VAR CONSTANT
	    CstClockReadTime 		: LTIME := LTIME#1S;	  				// (Time) Read Modbus Frequency .	
END_VAR

METHOD M_Execute
//////////////////
//  Method Calls 
/////////////////

VAR 
	// Method local variables (reinitialized at each cycle) 

END_VAR
SUPER^.M_Execute();
END_METHOD

END_FUNCTION_BLOCK

// ---- 01_Equipement_Library/ProtectRelay/FB_ProtectRelay_SepamS48.TcPOU
FUNCTION_BLOCK FB_ProtectRelay_SepamS48 EXTENDS FB_ProtectRelay_Base
//////////////////
// SEPAM system for High Voltage or Low Voltage Grid Protection. 
//////////////////

VAR_INPUT PERSISTENT
	// Parameters of the Object (instance/model specific) 
	   ParamTimeoutRTU						: TIME  := T#10S;					(* (s)	  Com RTU Timeout *)
	   ParamUnitID							: BYTE 	:= 1;						(* (NA)	  unit ID*)
	   ParamInInterfaceSub					: BOOL;								(* (NA)   Serial interface RS422/RS485 TYPE (0:EL6021, 1:SUB9)*)
END_VAR

VAR_OUTPUT
	//Child objects
	OUT_Protect_GTE_LONG_Running			: BOOL; 							// Long GTE fault, PP stop for 2m and lost of autorisation 

END_VAR

VAR_INPUT
	// I/O Inputs	
	IN_MesAlarmIMax_IO						: BOOL; 							// I max fault Fault, Losing autorisation and not possible to consumed
	IN_MesAlarmUmin_IO						: BOOL; 							// U min Fault, Keeping autorisation, If we have 3 gte in 30 min ==> Stop fedding and consumed during 2h
	IN_MesAlarmPWH_IO						: BOOL; 							// Defaut wattmétrique
	                                                								                                                	
	IN_CmdReset_3GTEFault					: BOOL; 							// 3GTE Fault Reset 
		
END_VAR

VAR
	//M_Read
	Trig_Read								: R_TRIG;
	ModbusRTU								: FB_ModbusRTU ;					// (NA) FB for Modbus Reading
	MbStruct								: ARRAY[1..2] OF Struct_InputRTU;

                                			
	ModbusAlarm								: ARRAY[1..2] OF BOOL;					// (NA) Read alarm
	AX_Quantity								: ARRAY[1..2] OF WORD;					// (NA) Quantity of blocks to read
	AX_Address								: ARRAY[1..2] OF WORD;					// (NA) Start address of the read
	OutErrorMbRead							: ARRAY[1..2] OF BOOL;
                                			
	Busy									: BOOL;
	MesBlock_Temp							: ARRAY [1..2] OF ARRAY [0..94] OF WORD;
	                            			
	RTrigI									: R_TRIG;
MesDataExd					AT %Q* 		: ProtectRelay_S48  ; 
	                            			
	//M_EVALUATE                			
	TON_GteIsLong							: TON;


		
END_VAR

METHOD M_Execute
//////////////////
//  Method Calls 
/////////////////

VAR 
	// Method local variables (reinitialized at each cycle) 
	MesStateCB	 : BOOL;

	KK 			 : INT;
	CalNbFeederClosed	: UINT ; 
END_VAR



CalNbFeederClosed := 0 ; 
FOR KK:= 1 TO CstNbFeederMVCB_G DO 
	CalNbFeederClosed :=  CalNbFeederClosed + SEL(A1_SUBMV.AX_FeederMVCB[KK].MesClosed , 0, 1 ) ; 

END_FOR




	
MesStateCB := A1_SUBMV.A1_MainMVCB.MesDataExd.MesData.MesClosed;
MesDataExd.MesData.MesI1 := 0;

IF MesStateCB THEN
	FOR KK:=1 TO CstNbPTR_G DO
	MesDataExd.MesData.MesI1 := MesDataExd.MesData.MesI1 + AX_PTR[KK].MesDataExd.MesData.MesI;
	END_FOR  
	

MesDataExd.MesData.MesI1 := MesDataExd.MesData.MesI1 *CalNbFeederClosed /CstNbFeederMVCB_G;
		

	
MesDataExd.MesData.MesI2 	:= MesDataExd.MesData.MesI1 ; 	
MesDataExd.MesData.MesI3 	:= MesDataExd.MesData.MesI1 ; 
MesDataExd.MesData.MesI0 	:= 0 ;
 
ELSE 
MesDataExd.MesData.MesI1 	:= 0 ;
MesDataExd.MesData.MesI2 	:= 0 ;
MesDataExd.MesData.MesI3 	:= 0 ;
MesDataExd.MesData.MesI0 	:= 0 ;
END_IF

MesDataExd.MesData.MesImax1	:= MAX(MesDataExd.MesData.MesImax1 , MesDataExd.MesData.MesI1  ) ; 
MesDataExd.MesData.MesImax2	:= MAX(MesDataExd.MesData.MesImax2 , MesDataExd.MesData.MesI2  ) ; 
MesDataExd.MesData.MesImax3	:= MAX(MesDataExd.MesData.MesImax3 , MesDataExd.MesData.MesI3  ) ; 
MesDataExd.MesData.MesImax0	:= MAX(MesDataExd.MesData.MesImax0 , MesDataExd.MesData.MesI0  ) ; 

MesDataExd.MesData.MesU12:= A1_SUBMV.MesDataExd.MesData.MesU;
MesDataExd.MesData.MesU31:= MesDataExd.MesData.MesU12;
MesDataExd.MesData.MesU23:= MesDataExd.MesData.MesU12;

MesDataExd.MesV1 := MesDataExd.MesData.MesU12/SQRT(3) ;
MesDataExd.MesV2 := MesDataExd.MesV1;	 
MesDataExd.MesV3 := MesDataExd.MesV1;

MesDataExd.MesData.MesFreq := A1_SUBMV.MesDataExd.MesData.MesFreq;
MesDataExd.MesP := A1_SUBMV.MesDataExd.MesData.MesPsol ; // Psol - Pload - Paux 
MesDataExd.MesQ := A1_SUBMV.MesDataExd.MesData.MesQsol; 
MesDataExd.MesS := SQRT(MesDataExd.MesP* MesDataExd.MesP + MesDataExd.MesQ*MesDataExd.MesQ);
MesDataExd.MesCosPhi := MesDataExd.MesP / MesDataExd.MesS;

IF MesDataExd.MesP > 0 THEN
	MesDataExd.EActProd := MesDataExd.EActProd + MesDataExd.MesP*ParamCycleTime_Emul/3600000	;
END_IF
IF MesDataExd.MesP < 0 THEN
	MesDataExd.EActCons := MesDataExd.EActCons - MesDataExd.MesP*ParamCycleTime_Emul/3600000	;
END_IF
IF MesDataExd.MesQ > 0 THEN
	MesDataExd.EReactProd := MesDataExd.EReactProd + MesDataExd.MesQ*ParamCycleTime_Emul/3600000	;
END_IF
IF MesDataExd.MesQ < 0 THEN
	MesDataExd.EReactCons := MesDataExd.EReactCons - MesDataExd.MesQ*ParamCycleTime_Emul/3600000	;
END_IF
END_METHOD

END_FUNCTION_BLOCK

// ---- 01_Equipement_Library/ProtectRelay/FB_ProtectRelay_SepamT20.TcPOU
FUNCTION_BLOCK FB_ProtectRelay_SepamT20 EXTENDS FB_ProtectRelay_Base
//////////////////
// SEPAM system for High Voltage or Low Voltage Grid Protection . 
//////////////////
VAR_INPUT PERSISTENT
	// Parameters of the Object (instance/model specific) 
	 
END_VAR

VAR_OUTPUT
	//Child objects
	OutFBCompleteted						: BOOL;
END_VAR

VAR_INPUT
	InUnitID            : DINT;			// (NA)   ID FOR SEPAM T20 Modbus Unit ID. 

	// I/O Inputs		
END_VAR

VAR
	//M_Read
	FB_ModbusRead_I1						: FB_ReadModbusRTU_V2; 				// (NA) FB for Modbus Reading
	FB_ModbusRead_I2						: FB_ReadModbusRTU_V2; 				// (NA) FB for Modbus Reading
	FB_ModbusRead_I3						: FB_ReadModbusRTU_V2; 				// (NA) FB for Modbus Reading
	ParamTimeoutRTU							: TIME:=T#10S;
	MesBlock1_Temp							: ARRAY [0..36] OF WORD;
	MesBlock2_Temp							: WORD;
	MesBlock3_Temp							: WORD;
	MesModbusAlarmCode						: UDINT;							// (NA) Modbus Read Alarm Code
	MesModbusAlarmCode2						: UDINT;							// (NA) Modbus Read Alarm Code
	MesModbusAlarmCode3						: UDINT;							// (NA) Modbus Read Alarm Code
	ModbusReadAlarm 						: BOOL;								// (NA) Modbus Read Alarm for communications
	ModbusReadAlarm2 						: BOOL;	
	ModbusReadAlarm3 						: BOOL;	
	AX_bRead 								: ARRAY [1..3] OF BOOL;
	CalAllCompleted							: BOOL;
	//M_ALARMMANAGEMENT VARIABLES//

	//M_Execute
	AllNotBusy								: BOOL;
	TP_Read									: TP;
	RTrig									: R_TRIG;
//	ClockRead								: BOOL;
	
	//EValuate//
MesDataExd					AT %Q* 		: ProtectRelay_T20;
	

		
END_VAR

METHOD M_Execute
//////////////////
//  Method Calls 
/////////////////

VAR 
	// Method local variables (reinitialized at each cycle) 

END_VAR
SUPER^.M_Execute();
END_METHOD

END_FUNCTION_BLOCK

// ---- 01_Equipement_Library/ProtectRelay/FB_ProtectRelay_VIP410.TcPOU
FUNCTION_BLOCK FB_ProtectRelay_VIP410 EXTENDS FB_ProtectRelay_Base
//////////////////
// SEPAM system for High Voltage or Low Voltage Grid Protection . 
//////////////////
VAR_INPUT PERSISTENT
	ParamTcpPort				: UINT:=502;    // (NA) TCP port
	ParamIPAddress				: STRING; 		// (NA) IP address
	ParamUnitID					: BYTE; 		// (NA) unit ID
END_VAR

VAR_OUTPUT
	
END_VAR

VAR_INPUT
		IN_MesTrip_IO			: BOOL ; 
END_VAR

VAR
	
	MesDataExd		AT %Q* 		: ProtectRelay_VIP410;
	FB_ModbusRead	          	: ARRAY[1..4] OF FB_ModbusRead; 
	ClockReadInput				: BOOL;

	MesBlock1_Temp 				: ARRAY [1..1] OF WORD ; 
	MesBlock2_Temp 				: ARRAY [1..20] OF WORD ; 
	MesBlock3_Temp 				: ARRAY [1..8] OF WORD ; 
	MesBlock4_Temp 				: ARRAY [1..2] OF WORD ; 
	AX_ModbusReadAlarm			: ARRAY[1..4] OF BOOL;
	AX_ModbusReadAlarmId		: ARRAY[1..4] OF UDINT;	
//	TP1							: TP ; 				// (NA) Tempo to define Modbus Reading Frequency 
	ParamClockInputTime 		: TIME 		:= TIME#5S;	  		// (Time) Read Modbus Frequency . 
END_VAR

METHOD M_Execute
//////////////////
//  Method Calls 
/////////////////

VAR 
	// Method local variables (reinitialized at each cycle) 

END_VAR
SUPER^.M_Execute();
END_METHOD

END_FUNCTION_BLOCK

// ---- 01_Equipement_Library/ProtectRelay/FB_ProtectRelay_WIP1.TcPOU
FUNCTION_BLOCK FB_ProtectRelay_WIP1 EXTENDS FB_ProtectRelay_Base
VAR_INPUT
						
	
	

END_VAR

VAR_INPUT
	// I/O Inputs 		                                     				
		IN_MesAlarmImax_IO		: BOOL ; // IO max I  fault
		IN_MesAlarmUmin_IO		: BOOL ;  // IO Min U  Fault 
		
END_VAR


VAR
// M_ALARMMNGMT VARIABLES //
                            		
	CmdResetHVCell				: BOOL ; 
	// M_READ VARIABLES//
	
MesDataExd 		    AT %Q*  	: ProtectRelay_WIP1; 	
		


END_VAR

METHOD M_Execute
SUPER^.M_Execute();
END_METHOD

END_FUNCTION_BLOCK

// ---- 01_Equipement_Library/Router/FB_Router.TcPOU
FUNCTION_BLOCK FB_Router

VAR_INPUT PERSISTENT 
	ParamTempoRestart	: TIME 		:= T#30S ;	//  (s)Tempo to wait before resupplying the ADSL routeur

	
END_VAR

        	
VAR_INPUT           	
	Heure_Local     	: TIMESTRUCT;
	IN_CmdRestart 			: BOOL;

	
	IN_CmdReset_L			: BOOL ;	// (NA) External Reset Command
	
END_VAR     


VAR_OUTPUT
	//Child objects
		OUT_CmdOpen_IO			: BOOL;	
END_VAR        	
      	
VAR                 	
	bInit				: BOOL;	// Booleen d'initialisation
		
	TP_Restart			: TP;
	// State Mananger //
	
	MesState			: BYTE; // Cal
MesDataExd			: Router_Standard;
	// M_Evaluate //
	
END_VAR

METHOD M_Execute : BOOL
VAR_INPUT
END_VAR
END_METHOD

END_FUNCTION_BLOCK

// ---- 01_Equipement_Library/Sensors/ANA/FB_ANA_Base.TcPOU
FUNCTION_BLOCK FB_ANA_Base 
//////////////////
// Analogic sensor . Base FB . 
//////////////////

VAR_INPUT PERSISTENT
	// Parameters of the Object (instance/mùodel specific) 
	ParamVarMaxAlarm		: REAL 		:=105		; // (%)  Config : Maximal allowed Site Hygrometry 
	ParamVarMaxWarning		: REAL 		:=90		; // (%)  Config : Maximal Site hygrometry warning
	ParamVarMinAlarm		: REAL 		:=-5		; // (%)  Config : Minimal allowed Site Hygrometry 
	ParamVarMinWarning		: REAL 		:=0			; // (%)  Config : Minimal Site hygrometry warning
	ParamDiffMax			: REAL 		:= 20 ; 	; // (NA) Config : Maximal Analogic difference acceptable between two sensors
	
	ParamNbSensors			: INT 		:=1			; // (NA) Config : Number of sensors
	
END_VAR

VAR_OUTPUT
	//Child objects
	
END_VAR

VAR_INPUT
	// I/O Inputs 
		IN_MesValue1_IO					: INT ; 	// 	IO Value
		IN_MesValue2_IO					: INT ; 	// 	IO Value

		IN_MesVar1Fault_IO		AT %I*		: BOOL ; 		 	//(NA)  sensor 1 has a 0 mA fault . 
		IN_MesVar2Fault_IO				: BOOL ; 		 	//(NA)  sensor 2 has a 0 mA fault . 		
END_VAR

VAR
	//M_ALARMMANAGEMENT VARIABLES//

		RS_MaxAlarm: RS;
		RS_MinAlarm: RS;
		RS_MinWarning: RS;
		RS_MaxWarning: RS;
	
		RSDiff: RS;
                                         	
	//M_READ VARIABLES//
		MesValue1						: REAL ;  	// temporary Value
		MesValue2						: REAL ; 
		
//	MesDataExd					: ANA ; 
	//EMULATOR //
		
		// M_INIT //
		bInit 						: BOOL;
		IN_CmdReset_L					: BOOL;
END_VAR

METHOD M_Execute
//////////////////
//  Method Calls 
/////////////////

VAR 
	// Method local variables (reinitialized at each cycle) 

END_VAR
END_METHOD

END_FUNCTION_BLOCK

// ---- 01_Equipement_Library/Sensors/ANA/FB_ANA_IO.TcPOU
FUNCTION_BLOCK FB_ANA_IO EXTENDS FB_ANA_Base
//////////////////
// Analogic sensor . Base FB . 
//////////////////

VAR_INPUT PERSISTENT
	// Parameters of the Object (instance/mùodel specific) 
		ParamName				: STRING:='TempPcs' ;			// (NA) Name of the pyranometer : to easily identify it
		ParamScaleMin			: REAL:=4 ; 		// (NA) minimal input value . 
		ParamScaleMax			: REAL:=20 ; 		// (NA) maximal input value .
		ParamRangeMin			: REAL:=0 ; 		// (NA) minimal output value . Unit depends on output 
		ParamRangeMax			: REAL:=100 ; 		// (NA) maximal output value . Unit depends on output 

		
		ParamForced_4_20		: BOOL:=FALSE;		// Is the input between 4-20mA ? 
		ParamPT100				: BOOL:=FALSE;	// IF PT 100
		ParamFix				: INT:=1 ; // Value to wich divide the initial value 
END_VAR

VAR_OUTPUT
	//Child objects
	
END_VAR

VAR_INPUT
	// I/O Inputs 
		//MesIO1							: INT ; 	// 	IO Value
		IN_MesIOReal1						: REAL;
		IN_MesIOReal2						: REAL;
		
END_VAR

VAR
	//M_ALARMMANAGEMENT VARIABLES//
              MesData			: ANA ;     	
	//M_READ VARIABLES//


		
END_VAR

END_FUNCTION_BLOCK

// ---- 01_Equipement_Library/Sensors/ANA/FB_ANA_Irra_Fx.TcPOU
FUNCTION_BLOCK FB_ANA_Irra_Fx EXTENDS FB_ANA_Base
//////////////////
// (4-20 mA) sensor . 
//////////////////

VAR_INPUT PERSISTENT
	// Parameters of the Object (instance/model specific) 
	ParamSensibility				: REAL ;			// Sensibility of the sensor ? 
END_VAR

VAR_OUTPUT
	//Child objects
	
END_VAR

VAR_INPUT
	// I/O Inputs 
	
END_VAR         			
                			
VAR             			
	A						: REAL;     // F(x) = Ax+B
	B						: REAL;     // F(x) = Ax+B

	 MesData			: ANA ;   
		
END_VAR

METHOD M_Execute
//////////////////
//  Method Calls 
/////////////////

VAR 
	// Method local variables (reinitialized at each cycle) 

END_VAR


SUPER^.M_Execute() ;
END_METHOD

END_FUNCTION_BLOCK

// ---- 01_Equipement_Library/Sensors/COM/FB_AllInOne.TcPOU
FUNCTION_BLOCK FB_AllInOne
VAR_INPUT
	ParamNameAllInOne		: STRING 	:= 'Wind spd + dir + hygro + temp';				// (NA) Name of the pyranometer : to easily identify it
	ParamTempoComAlarm		: TIME 		:= T#10S ; 										// (s) Config : Tempo to detect LOC Alarm
	ParamClockReadTime 		: TIME 		:= T#2S;	  									// (Time) Read Modbus Frequency . 
 	ParamTimeout			: TIME  	:= T#5S ;		  								// (Time) Timeout for modbus reading
	ParamUnitID				: BYTE		:= 1;											// (NA) Unit ID for modbus reading
	ParamTCPPort			: UINT		:= 502;											// (NA) TCP port for modbus
	ParamIpAddress			: STRING	:= '127.0.0.1';									// (NA) IP address for modbus
END_VAR

VAR
	//M_AlarmManagement
	TON_ComAlarm				: TON ; 						// Tempo before deteting loss of communication. 

	
	IN_CmdReset_L					: BOOL;                                                        	
		
	// M_READ VARIABLES//
MesData		AT %Q*  : AllInOne ; 							// (NA) [P,H,B] INV  Data Structure 
	FB_ModbusReadInputRegs		: ARRAY[1..2] OF FB_MBReadInputRegs;		// FB for Modbus Read
	MesBlock1_Temp 				: ARRAY[1..96]  OF WORD; 		// (NA) Temporary Block with multiple modbus reading (Caution : Double Word variables)
	MesBlock2_Temp 				: ARRAY[1..3]  OF WORD; 		// (NA) Temporary Block with multiple modbus reading (Caution : Double Word variables)
	MesModbusReadAlarm1 		: BOOL ; 						// (NA) Modbus Read Alarm for all modbus frames		
	MesModbusReadAlarm2 		: BOOL ; 						// (NA) Modbus Read Alarm for all modbus frames		
	MesAlarmCom					: BOOL;
	MesModbusAlarmCode			: UDINT;						// (NA) Modbus Read Alarm Code	
	
	// M_STATEMANAGER//
	FB_OperationIndex			: FB_OperationIndex ; 
	CalLastStart				: STRING ;			 			// Datetime of the last Start
	MesState					: BYTE ; 						// (NA) Cal                                                                                                            	
	CalRunningTime				: INT ; 						// Total Running Time
	                                                        	
	//M_EXECUTE VARIABLES //                                	
	TP1							: TP ; 							// (NA) Tempo to define Modbus Reading Frequency 
	                                                        	
	ClockRead					: BOOL;							// (NA) Modbus reading Clock
	
	
	//M_INIT //
	bInit 						: BOOL;							 
END_VAR

VAR_OUTPUT
END_VAR
VAR
END_VAR

METHOD M_Execute
//////////////////
//  Method Calls 
/////////////////

VAR 
	// Method local variables (reinitialized at each cycle) 

END_VAR
END_METHOD

END_FUNCTION_BLOCK

// ---- 01_Equipement_Library/Sensors/COM/FB_ANA_SMP1X.TcPOU
FUNCTION_BLOCK FB_ANA_SMP1X
VAR_INPUT PERSISTENT
	
	ParamNamePyranometer	: STRING 	:= 'Wind spd + dir + hygro + temp + pluvio';	// (NA) Name of the eqt : to easily identify it
	ParamTempoComAlarm		: TIME 		:= T#10S ; 										// (s) Config : Tempo to detect LOC Alarm
	ParamClockReadTime 		: TIME 		:= TIME#1S;	  									// (Time) Read Modbus Frequency . 
 	ParamTimeout			: TIME  	:= T#2S ;		  								// (Time) Timeout for modbus reading
	ParamUnitID				: BYTE		:= 1;											// (NA) Unit ID for modbus reading
	
END_VAR

VAR
	//M_AlarmManagement
	TON_ComAlarm				: TON ; 						// Tempo before deteting loss of communication. 

	MesAlarmCom					: BOOL;
	
	IN_CmdReset_L					: BOOL;                                                        	

	
	// M_READ VARIABLES//
		MesDataExd.MesData	AT %Q*	      	: SMP1X ; 					// (NA) [P,H,B] INV  Data Structure 
	//ModbusRead_RTU				: FB_ReadModbusRTU_V2;			// FB for Modbus Read
	bReadError					: BOOL;
	bReadCompleted 				: BOOL;
	bReadBusy					: BOOL;
	InputStructRead 			: Struct_InputRTU;
	
	MesBlock1_Temp 				: ARRAY[1..125]  OF WORD; 		// (NA) Temporary Block with multiple modbus reading (Caution : Double Word variables)
	MesModbusReadAlarm 		  	: BOOL ; 						// (NA) Modbus Read Alarm for all modbus frames		
	MesModbusAlarmCode			: UDINT;						// (NA) Modbus Read Alarm Code	
	
	ScaleFactor					: REAL;
	BodyTemp					: REAL;
	StatusFlag					: REAL;
	
	// M_STATEMANAGER//
	FB_OperationIndex			: FB_OperationIndex ; 
	CalLastStart				: STRING ;			 			// Datetime of the last Start
	MesState					: BYTE ; 						// (NA)                                                                                                            	
	CalRunningTime				: INT ; 						// Total Running Time
	                                                        	
	//M_EXECUTE VARIABLES //                                	
	TP1							: TP ; 							// (NA) Tempo to define Modbus Reading Frequency 
	                                                        	
	ClockRead					: BOOL;							// (NA) Modbus reading Clock
	
	
	//M_INIT //
	bInit 						: BOOL;							 
END_VAR

VAR_OUTPUT
END_VAR
VAR
END_VAR

METHOD M_Execute
//////////////////
//  Method Calls 
/////////////////

VAR 
	// Method local variables (reinitialized at each cycle) 

END_VAR
END_METHOD

END_FUNCTION_BLOCK

// ---- 01_Equipement_Library/Sensors/TOR/FB_TOR_Base.TcPOU
FUNCTION_BLOCK FB_TOR_Base
//////////////////
//  Digital SensOR  Base FB . 
//////////////////

VAR_INPUT PERSISTENT
	// Parameters of the Object (instance/model specific) 
	ParamNbSensors			: INT 		:=1			; // (NA) Config : Number of sensors, If =9 Then sensor is bi-stable contactOR 
	ParamAtleastOne			: BOOL 		:= TRUE ;  // If TRUE, the output is true if at leat one of the sensor is active. Otherwise , the output is true only if both are active
	ParamCableCutSecurity	: BOOL		:=FALSE;	// FALSE = ALARM ; 
	
	CalCountAlarm			: UDINT 	:=0 ; // Count number of times the alarm has been triggered.
	
END_VAR

VAR_OUTPUT
	//Child objects
	
END_VAR

VAR_INPUT
	// I/O Inputs 		                                     				
		IN_MesState1_IO 					: BOOL;	 				// (NA) First  Smoke detector IO, IF bi-stable NC
		IN_MesState2_IO					: BOOL ; 				// (NA) Second Smoke detector IO, IF Bi-stable NO
		IN_CmdReset_L					: BOOL;				// LOCAL Reset Value For Alarms
		IN_ResetCounter 				: BOOL ; 			// Reset counter . 
END_VAR

VAR
	//M_ALARMMANAGEMENT VARIABLES//

	//STATE MANAGEMENT //
//	MesDataExd				: TOR ; 	
		R_TRIGAlarm					: R_TRIG  ; 

	// EMULATOR 
	
END_VAR

METHOD M_Execute
//////////////////
//  Method Calls 
/////////////////

VAR 
	// Method local variables (reinitialized at each cycle) 
	
END_VAR
END_METHOD

END_FUNCTION_BLOCK

// ---- 01_Equipement_Library/Sensors/TOR/FB_TOR_CB.TcPOU
FUNCTION_BLOCK FB_TOR_CB EXTENDS FB_TOR_Base
//////////////////
//  Door sensor system . State = True >> Door Closed .
//////////////////

VAR_INPUT PERSISTENT
	// Parameters of the Object (instance/model specific) 
		
		
END_VAR

VAR_OUTPUT
	//Child objects
	
END_VAR

VAR_INPUT
	// I/O Inputs 		                                     				
		
END_VAR

VAR
	//M_ALARMMANAGEMENT VARIABLES//
		
MesDataExd			: TOR_Standard ;  

	
END_VAR

END_FUNCTION_BLOCK

// ---- 01_Equipement_Library/Sensors/TOR/FB_TOR_DS.TcPOU
FUNCTION_BLOCK FB_TOR_DS EXTENDS FB_TOR_Base
//////////////////
//  Door sensor system . State = True >> Door Closed .
//////////////////

VAR_INPUT PERSISTENT
	// Parameters of the Object (instance/model specific) 
		ParamTempoDoorAlarm			: TIME := T#10S ;	// (s) Tempo for Door sensor alarm 
		
END_VAR

VAR_OUTPUT
	//Child objects
	
END_VAR

VAR_INPUT
	// I/O Inputs 		                                     				
		
END_VAR

VAR
	//M_ALARMMANAGEMENT VARIABLES//
		TON_Ouverture				: TON;				//(NA) Tempo to detect door opened for too long time . 
	MesDataExd			: TOR_Standard ;  



END_VAR

METHOD M_Execute
//////////////////
//  Method Calls 
/////////////////

VAR 
	// Method local variables (reinitialized at each cycle) 
	
END_VAR


SUPER^.M_Execute() ;
END_METHOD

END_FUNCTION_BLOCK

// ---- 01_Equipement_Library/Sensors/TOR/FB_TOR_ES.TcPOU
FUNCTION_BLOCK FB_TOR_ES EXTENDS FB_TOR_Base
//////////////////
//  Emergency stop system
//////////////////
VAR_INPUT PERSISTENT
	// Parameters of the Object (instance/model specific) 
	ParamTempoEs :TIME:=T#2S;	// (s) Tempo before raising an alarm
END_VAR

VAR_OUTPUT
	//Child objects
	
END_VAR

VAR_INPUT
	// I/O Inputs 		                                     				
		
	
END_VAR

VAR
	//M_ALARMMANAGEMENT VARIABLES//
		FB_PermAlarm				: SR ;					// (NA) FB to maintain emergency stop Alarm 
		TON_ES						: TON ; 
 
	//M_STATEMANAGER VARIABLES//
		MesDataExd			: TOR_Standard ;  	
	// EMULATOR //
		Emul_MesState1				: BOOL;
		Emul_MesState2				: BOOL;
		
END_VAR

METHOD M_Execute
//////////////////
//  Method Calls 
/////////////////

VAR 
	// Method local variables (reinitialized at each cycle) 

END_VAR

	
	IF ParamNbSensors = 9 THEN // Use of contactor bi-stable No and NC
		IN_MesState2_IO := NOT IN_MesState2_IO;
	END_IF
SUPER^.M_Execute() ;
END_METHOD

END_FUNCTION_BLOCK

// ---- 01_Equipement_Library/Sensors/TOR/FB_TOR_Fuse.TcPOU
FUNCTION_BLOCK FB_TOR_Fuse EXTENDS FB_TOR_Base
//////////////////
//  Smoke and Fire detection system with Typhoon triggering system. 
//////////////////
VAR_INPUT PERSISTENT
	// Parameters of the Object (instance/model specific) 
	ParamTempoFuse :TIME:=T#5S;//  (s)Tempo before raising an alarm
END_VAR

VAR_OUTPUT
	//Child objects
	
END_VAR

VAR_INPUT
	// I/O Inputs 		                                     				
		
	
END_VAR

VAR
	//M_ALARMMANAGEMENT VARIABLES//
		FB_PermAlarm				: SR ;					// (NA) FB to maintain Fire Alarm even if sensor stop detection (burn) .
 		TON_Fuse					: TON; 	
	//M_STATEMANAGER VARIABLES//
	MesDataExd			: TOR_Standard ;  

		
END_VAR

METHOD M_Execute
//////////////////
//  Method Calls 
/////////////////

VAR 
	// Method local variables (reinitialized at each cycle) 

END_VAR
// EMULATOR I/O //

	
	IF ParamNbSensors = 9 THEN // Use of contactor bi-stable No and NC
		IN_MesState2_IO := NOT IN_MesState2_IO;
	END_IF
SUPER^.M_Execute() ;
END_METHOD

END_FUNCTION_BLOCK

// ---- 01_Equipement_Library/Sensors/TOR/FB_TOR_MS.TcPOU
FUNCTION_BLOCK FB_TOR_MS EXTENDS FB_TOR_Base
//////////////////
//  Door sensor system . State = True >> Door Closed .
//////////////////

VAR_INPUT PERSISTENT
	// Parameters of the Object (instance/model specific) 
		ParamTempoDoorAlarm			: TIME := T#10S ;	// (S) Tempo for Door sensor alarm 
		
END_VAR

VAR_OUTPUT
	//Child objects
	
END_VAR

VAR_INPUT
	// I/O Inputs 		                                     				
		
END_VAR

VAR
	//M_ALARMMANAGEMENT VARIABLES//
		TP_Fermeture			: TP;				//(NA) Tempo to detect door opened for too long time . 
		RS_fermeture			: RS;
		
		MesDataExd			: TOR_Standard ;  
		


END_VAR

METHOD M_Execute
//////////////////
//  Method Calls 
/////////////////

VAR 
	// Method local variables (reinitialized at each cycle) 
	
END_VAR

SUPER^.M_Execute() ;
END_METHOD

END_FUNCTION_BLOCK

// ---- 01_Equipement_Library/Sensors/TOR/FB_TOR_Rain.TcPOU
FUNCTION_BLOCK FB_TOR_Rain EXTENDS FB_TOR_Base
//////////////////
//  Door sensor system . State = True >> Door Closed .
//////////////////

VAR_INPUT PERSISTENT
	// Parameters of the Object (instance/model specific) 
	
		
END_VAR

VAR_OUTPUT
	//Child objects
	
END_VAR

VAR_INPUT
	// I/O Inputs 		                                     				
	
    ParamVarHrWarning   : REAL:=8;  // Max of raining before warning mm of rain for last hour --> Mean it is raining a lot  Defaut value 8       
    ParamVarDayWarning  : REAL:=48; // max of raining before warning mm of rain for last day  --> Mean it rained a lot during 1 day defaut value 48
	ParamVarMinAlarm	: REAL 	:=-5		; // (%)  Config : Minimal allowed Site Hygrometry 
	
END_VAR

VAR
	MesDataExd			: TOR_Rain;

	//M_ALARMMANAGEMENT VARIABLES//
		WarningDay					: BOOL;
		WarningHr					: BOOL;
		WarningValue				: BOOL;
	
	//GET/SET PROPERTY MANAGEMENT//
	//M_Execute
		FB_AverageHr				: FB_Average; 	
	    FB_AverageDay               : FB_Average;
	    FB_AverageMonth             : FB_Average;
		CTUHr						: CTU;
		CTUDay						: CTU;
		CTUMonth					: CTU;
		Hour 						: INT;
		PluvioHr_Avg		        : REAL ; 
		PluvioDay_Avg		        : REAL ; 
		PluvioMonth_Avg		        : REAL ;     
		PluvioHr_Max		        : REAL;
		PluvioDay_Max		        : REAL ; 
		PluvioMonth_Max		        : REAL ; 
        PluvioHr					: REAL ; 
		PluvioDay					: REAL ; 
		PluvioMonth					: REAL ; 

	
	
END_VAR

METHOD M_Execute
//////////////////
//  Method Calls 
/////////////////

VAR 
	// Method local variables (reinitialized at each cycle) 
	
END_VAR
// EMULATOR I/O //

//MAIN CODE HERE
Hour 							:=CstCycleTime_G/1000/3600  ;                        

CTUHr   (CU:= MesDataExd.MesData.MesAlarmState , RESET :=  Hour MOD 1 = 0) ; 
CTUDay  (CU:= MesDataExd.MesData.MesAlarmState , RESET := Hour MOD 24 = 0 ) ; 
CTUMonth(CU:= MesDataExd.MesData.MesAlarmState , RESET := Hour MOD 24*30 = 0 ) ; 

PluvioHr_Max := SEL( Hour MOD 1 = 0  ,   PluvioHr_Max , PluvioHr_Max:= PluvioHr)  ; 
PluvioHr := CTUHr.CV  ; 

PluvioDay_Max := SEL( Hour MOD 24 = 0  ,   PluvioDay_Max , PluvioDay_Max:= PluvioDay)  ; 
PluvioDay := CTUDay.CV  ; 

PluvioMonth_Max := SEL( Hour MOD 24*30 = 0  ,   PluvioMonth_Max , PluvioMonth_Max:= PluvioMonth)  ; 
PluvioMonth := CTUMonth.CV  ; 


FB_AverageHr(ValueIn:=PluvioHr_Max  , WindowDuration := 24*3600*1000 , ValueOut => PluvioHr_Avg) ; 
FB_AverageDay(ValueIn:=PluvioDay_Max  , WindowDuration := 24*30*3600*1000 , ValueOut => PluvioDay_Avg) ; 
FB_AverageMonth(ValueIn:=PluvioMonth_Max  , WindowDuration := 24*365*3600*1000 , ValueOut => PluvioMonth_Avg) ;
//EVALUATE

MesDataExd.MesRainFall_LastHour 	:= PluvioHr;
MesDataExd.MesRainFall_LastDay		:= PluvioDay;
MesDataExd.MesRainFall_LastMonth	:= PluvioMonth;
MesDataExd.AvgmmHour		:= PluvioHr_Avg;
MesDataExd.AvgmmDay		:= PluvioDay_Avg;
MesDataExd.AvgmmMonth		:= PluvioMonth_Avg;


SUPER^.M_Execute();
END_METHOD

END_FUNCTION_BLOCK

// ---- 01_Equipement_Library/Sensors/TOR/FB_TOR_SD.TcPOU
FUNCTION_BLOCK FB_TOR_SD EXTENDS FB_TOR_Base
//////////////////
//  Smoke and Fire detection system with Typhoon triggering system. 
//////////////////
VAR_INPUT PERSISTENT
	// Parameters of the Object (instance/model specific) 
	ParamTempoFire :TIME:=T#2S;//  (s)Tempo before raising an alarm
END_VAR

VAR_OUTPUT
	//Child objects
	
END_VAR

VAR_INPUT
	// I/O Inputs 		                                     				
		
	
END_VAR

VAR
	//M_ALARMMANAGEMENT VARIABLES//
		FB_PermAlarm				: SR ;					// (NA) FB to maintain Fire Alarm even if sensor stop detection (burn) .
		TON_Fire					: TON ; 
 
	//M_STATEMANAGER VARIABLES//
		MesDataExd			: TOR_Standard ;  
		
		
END_VAR

METHOD M_Execute
//////////////////
//  Method Calls 
/////////////////

VAR 
	// Method local variables (reinitialized at each cycle) 

END_VAR

	IF ParamNbSensors = 9 THEN // Use of contactor bi-stable No and NC
		IN_MesState2_IO := NOT IN_MesState2_IO;
	END_IF
SUPER^.M_Execute() ;
END_METHOD

END_FUNCTION_BLOCK

// ---- 01_Equipement_Library/Sensors/TOR/FB_TOR_Spd.TcPOU
FUNCTION_BLOCK FB_TOR_Spd EXTENDS FB_TOR_Base
//////////////////
//  Smoke and Fire detection system with Typhoon triggering system. 
//////////////////
VAR_INPUT PERSISTENT
	// Parameters of the Object (instance/model specific) 
	ParamTempoEs :TIME:=T#5S;//  (s)Tempo before raising an alarm
END_VAR

VAR_OUTPUT
	//Child objects
	
END_VAR

VAR_INPUT
	// I/O Inputs 		                                     				
		
	
END_VAR

VAR
	//M_ALARMMANAGEMENT VARIABLES//
		FB_PermAlarm				: SR ;					// (NA) FB to maintain Fire Alarm even if sensor stop detection (burn) .
		TON_ES						: TON ; 
 
	//M_STATEMANAGER VARIABLES//
		MesDataExd			: TOR_Standard ;  

		
END_VAR

METHOD M_Execute
//////////////////
//  Method Calls 
/////////////////

VAR 
	// Method local variables (reinitialized at each cycle) 

END_VAR

	
	IF ParamNbSensors = 9 THEN // Use of contactor bi-stable No and NC
		IN_MesState2_IO := NOT IN_MesState2_IO;
	END_IF
SUPER^.M_Execute() ;
END_METHOD

END_FUNCTION_BLOCK

// ---- 01_Equipement_Library/Sensors/TOR/FB_TOR_Standard.TcPOU
FUNCTION_BLOCK FB_TOR_Standard EXTENDS FB_TOR_Base
//////////////////
//  Circuit Breaker
//////////////////

VAR_INPUT PERSISTENT
	// Parameters of the Object (instance/model specific) 
		
		
END_VAR

VAR_OUTPUT
	//Child objects
	
END_VAR

VAR_INPUT
	// I/O Inputs 		                                     				
		
END_VAR

VAR
	//M_ALARMMANAGEMENT VARIABLES//
		
MesDataExd			: TOR_Standard ;  

	
END_VAR

END_FUNCTION_BLOCK

// ---- 01_Equipement_Library/Sensors/TOR/FB_TOR_ToS.TcPOU
FUNCTION_BLOCK FB_TOR_ToS EXTENDS FB_TOR_Base
//////////////////
//  Technician on site selectOR   
//////////////////

VAR_INPUT PERSISTENT
	// Parameters of the Object (instance/model specific) 
	ParamTempoToSAlarm				: TIME := T#180M ; 	//(min) Tempo (2h30) after ToS without clear fault >> alarm 
	ParamTempoToSWarning			: TIME := T#120M ;  // (min) Tempo (2h) after ToS without clear fault  >> warning
END_VAR

VAR_OUTPUT
	//Child objects
	
END_VAR

VAR_INPUT
	// I/O Inputs 		                                     				
	
END_VAR

VAR
	//M_ALARMMANAGEMENT VARIABLES//
		TON 						: TON ;  			 // (NA) Calculate time since technician presence activation. 
		        
MesDataExd			: TOR_Standard ;                              			
	          	
	//GET/SET PROPERTY MANAGEMENT//
	
	//EMULATOR //
		Emul_MesState				: BOOL;
		
END_VAR

METHOD M_Execute
//////////////////
//  Method Calls 
/////////////////

VAR 
	// Method local variables (reinitialized at each cycle) 

END_VAR
// EMULATOR I/O //

SUPER^.M_Execute() ;
END_METHOD

END_FUNCTION_BLOCK

// ---- 01_Equipement_Library/Tariff Meter/FB_EM.TcPOU
FUNCTION_BLOCK FB_EM EXTENDS FB_EM_Base
//////////////////
// Measurement Solution. Base FB
//////////////////
VAR_INPUT PERSISTENT
	// Parameters of the Object (instance specific) 
		
	
END_VAR

VAR_OUTPUT
	//Child objects
	
END_VAR
VAR
	//M_ALARMMANAGEMENT VARIABLES//
		Eess: REAL;
	Eessinit	: REAL ; 
                             

	//M_INIT VARIABLES //
	
		
	// M_EXECUTE VARIABLES //
 		
	// M_Reset_L
		
                      
END_VAR

VAR_INPUT
		
END_VAR

METHOD M_Execute
//////////////////
//  Method Calls 
/////////////////
VAR 
	// Method local variables (reinitialized at each cycle) 
	// EMULATOR

	
END_VAR
Eess :=  Eess + ((A1_PP.MesDataExd.MesData.MesPbat + A1_SUBMV.MesDataExd.MesData.MesPaux)/6)*ParamCycleTime_Emul/3600000  ; 

MesPulseEactCons := FALSE ; 
IF Eess > Eessinit + ParamStepEactCons THEN	// every 10 kWh 
	MesPulseEactCons := TRUE ; 
	Eessinit := Eess ; 
END_IF
END_METHOD

END_FUNCTION_BLOCK

// ---- 01_Equipement_Library/Tariff Meter/FB_EM_Base.TcPOU
FUNCTION_BLOCK FB_EM_Base
//////////////////
// Measurement Solution. Base FB
//////////////////
VAR_INPUT PERSISTENT
	// Parameters of the Object (instance specific) 
		CmdInitialValues			: EM;
		ParamStepEactCons			: REAL := 10;					// kWh step for tariff meter
		ParamStepEactProd			: REAL := 10;                 // kWh step for tariff meter
		ParamStepEreactCons			: REAL := 10;                 // kVArh step for tariff meter
		ParamStepEreactProd			: REAL := 10;                 // kVArh step for tariff meter
		ParamEssNum					: UINT :=1 ; 					// ESS Num
END_VAR

VAR_INPUT
	//Child objects
		IN_CmdReset_L					: BOOL;													// (NA) Local reset of the alarms	
END_VAR
VAR
	//M_ALARMMANAGEMENT VARIABLES//
		TON_ComAlarm				: TON ; 												// Tempo before deteting loss of communication. 

	//M_INIT VARIABLES //
		bInit						: BOOL 				:= TRUE ; 							// (NA) Initialize object parameters at first cycle 
		
	// M_EXECUTE VARIABLES //
 //	MesDataExd			: EM;					// (NA) Structure of the Tariff Meter
		
	// M_EVALUATE VARIABLES //
		trig1 						: R_TRIG;												// (NA) Trigger for the pulses
		trig2 						: R_TRIG;												// (NA) Trigger for the pulses
		trig3 						: R_TRIG;												// (NA) Trigger for the pulses
		trig4 						: R_TRIG;												// (NA) Trigger for the pulses

                      
END_VAR

VAR_INPUT
		MesPulseEactCons			: BOOL;													// Pulse Input signal for the Active energy consumed measurement
		MesPulseEactProd			: BOOL;													// Pulse Input signal for the Active energy produced measurement
		MesPulseEreactCons			: BOOL;													// Pulse Input signal for the Reactive energy consumed measurement
		MesPulseEreactProd			: BOOL;													// Pulse Input signal for the Reactive energy produced measurement
END_VAR

METHOD M_Execute
//////////////////
//  Method Calls 
/////////////////
VAR 
	// Method local variables (reinitialized at each cycle) 
	// EMULATOR

	
END_VAR
END_METHOD

END_FUNCTION_BLOCK

// ---- 01_Equipement_Library/Tariff Meter/FB_EM_Pulse.TcPOU
FUNCTION_BLOCK FB_EM_Pulse EXTENDS FB_EM_Base
//////////////////
// Measurement Solution. Base FB
//////////////////
VAR_INPUT PERSISTENT
	// Parameters of the Object (instance specific) 
		
	
END_VAR

VAR_OUTPUT
	//Child objects
	
END_VAR
VAR
	//M_ALARMMANAGEMENT VARIABLES//
		FB_DetectFixedValue   : FB_DetectFixedValue ; 
        Eact_null    		  : REAL ;                                   								
		

	//M_INIT VARIABLES //
		MesDataExd			: EM_Standard ; 
		
	// M_EXECUTE VARIABLES //
 		
	// M_Reset_L
		
                      
END_VAR

VAR_INPUT
		
END_VAR

METHOD M_AlarmManagement
//////////////////
// Digiware measurement tool alarm and warning management
/////////////////

VAR 
	FB_AlarmCodeManager : FB_AlarmCodeManager ; 
END_VAR

FB_DetectFixedValue(IN_Addr := ADR(MesDataExd.MesData.MesEactCons) , IN_Size := SIZEOF(MesDataExd.MesData.MesEactCons) , IN_Duration :=T#3H , IN_EmptyStruct := ADR(Eact_null ) ); 

// ALARM CODE //
	FB_AlarmCodeManager(
		bAlarm1			:= MesDataExd.MesData.MesEActProd > 10 ,																			// Production measured			
		bAlarm2			:=FB_DetectFixedValue.OUT_bStatic 	,																	// Loss of communication with meter 
		bAlarm3			:=FALSE, 																								// 
		bAlarm4			:=FALSE, 																								// 
		bAlarm5			:=FALSE, 																								//
		bAlarm6			:=FALSE,        																						//
		bAlarm7			:=FALSE,        																						//
		bAlarm8			:=FALSE,        																						//
		bAlarm9			:=FALSE,        																						//
		bAlarm10		:=FALSE,        																						//
		bAlarm11		:=FALSE,        																						//
		bAlarm12		:=FALSE,        																						//
		bAlarm13		:=FALSE,        																						//
		bAlarm14		:=FALSE,        																						//
		bAlarm15		:=FALSE,        																						//
		wAlarmCode		=>MesDataExd.MesData.MesAlarmCode);

// WARNING CODE //

	FB_AlarmCodeManager(
		bAlarm1			:= FALSE ,										//  
		bAlarm2			:=FALSE, 										// 
		bAlarm3			:=FALSE, 										// 
		bAlarm4			:=FALSE, 										// 
		bAlarm5			:=FALSE, 										//
		bAlarm6			:=FALSE,        								//
		bAlarm7			:=FALSE,        								//
		bAlarm8			:=FALSE,        								//
		bAlarm9			:=FALSE,        								//
		bAlarm10		:=FALSE,        								//
		bAlarm11		:=FALSE,        								//
		bAlarm12		:=FALSE,        								//
		bAlarm13		:=FALSE,        								//
		bAlarm14		:=FALSE,        								//
		bAlarm15		:=FALSE,        								//
		wAlarmCode		=>MesDataExd.MesData.MesWarningCode);
			
// EVENT CODE //
	FB_AlarmCodeManager(
		bAlarm1			:= IN_CmdReset_L, 				// Reset command
		bAlarm2			:= FALSE, 						// 
		bAlarm3			:= FALSE, 						// 
		bAlarm4			:= FALSE, 						// 
		bAlarm5			:= FALSE, 						//
		bAlarm6			:= FALSE, 						//
		bAlarm7			:= FALSE,                       //
		bAlarm8			:= FALSE,                       //
		bAlarm9			:= FALSE,                       //
		bAlarm10		:= FALSE,                       //
		bAlarm11		:= FALSE,                       //
		bAlarm12		:= FALSE,                       //
		bAlarm13		:= FALSE,                       //
		bAlarm14		:= FALSE,                       //
		bAlarm15		:= FALSE,                       //
		wAlarmCode		=>MesDataExd.MesData.MesEventCode);
END_METHOD

METHOD M_Evaluate
VAR_INPUT
END_VAR

VAR
	TM_0 : EM_Standard;	// Empty structure
	OutTrig_Eac : BOOL;
	OutTrig_Eap : BOOL;
	OutTrig_Erc : BOOL;
	OutTrig_Erp : BOOL;
	bTest : BOOL;
END_VAR
IF CmdInitialValues.MesData.MesEactCons <> TM_0.MesData.MesEactCons OR CmdInitialValues.MesData.MesEActProd <> TM_0.MesData.MesEActProd OR CmdInitialValues.MesData.MesEReactCons <> TM_0.MesData.MesEReactCons OR CmdInitialValues.MesData.MesEReactProd <> TM_0.MesData.MesEReactProd THEN
MesDataExd:= CmdInitialValues;
	CmdInitialValues := TM_0 ;
END_IF

trig1(CLK := IN_MesPulseEactCons_IO, Q => OutTrig_Eac);
trig2(CLK := IN_MesPulseEactProd_IO, Q => OutTrig_Eap);
trig3(CLK:= IN_MesPulseEreactCons_IO, Q => OutTrig_Erc);
trig4(CLK:= IN_MesPulseEreactProd_IO, Q => OutTrig_Erp);

IF OutTrig_Eac THEN
MesDataExd.MesData.MesEactCons := MesDataExd.MesData.MesEactCons + ParamStepEactCons;
END_IF 

IF OutTrig_Eap THEN
MesDataExd.MesData.MesEActProd := MesDataExd.MesData.MesEActProd + ParamStepEactProd;
END_IF 

IF OutTrig_Erc THEN
MesDataExd.MesData.MesEReactCons := MesDataExd.MesData.MesEReactCons + ParamStepEreactCons;
END_IF 

IF OutTrig_Erp THEN
MesDataExd.MesData.MesEReactProd := MesDataExd.MesData.MesEReactProd + ParamStepEreactProd;
END_IF 

SUPER^.M_Evaluate();
END_METHOD

METHOD M_Init
VAR 
	InitialValues : EM_Standard ; 
END_VAR
MesDataExd := InitialValues ; 
bInit := FALSE ;
END_METHOD

END_FUNCTION_BLOCK

// ---- 01_Equipement_Library/Transfo/FB_Transfo_Base.TcPOU
FUNCTION_BLOCK FB_Transfo_Base
//////////////////
// High Voltage transformer with Transfo or DMCR detection . 
//////////////////

VAR_INPUT PERSISTENT
	// Parameters of the Object (instance/model specific) 

END_VAR

VAR_OUTPUT
	//Child objects
	
END_VAR

VAR_INPUT
		// Transfo

END_VAR

VAR
	//MesDataExd					: Transfo ; 
		
END_VAR

METHOD M_Execute
//////////////////
//  Method Calls 
/////////////////

VAR 
	// Method local variables (reinitialized at each cycle) 

END_VAR
END_METHOD

END_FUNCTION_BLOCK

// ---- 01_Equipement_Library/Transfo/FB_Transfo_HVCom.TcPOU
FUNCTION_BLOCK FB_Transfo_HVCom EXTENDS FB_Transfo_Base
//////////////////
// High Voltage transformer with Transfo or DMCR detection . 
//////////////////

VAR_INPUT PERSISTENT
	// Parameters of the Object (instance/model specific) 
	
END_VAR

VAR_OUTPUT
	//Child objects
	
END_VAR

VAR_INPUT

END_VAR

VAR
MesDataExd					: Transfo_HV ; 
		
END_VAR

END_FUNCTION_BLOCK

// ---- 01_Equipement_Library/Transfo/FB_Transfo_MV.TcPOU
FUNCTION_BLOCK FB_Transfo_MV EXTENDS FB_Transfo_Base
//////////////////
// High Voltage transformer with Transfo or DMCR detection . 
//////////////////

VAR_INPUT PERSISTENT
	// Parameters of the Object (instance/model specific) 

END_VAR

VAR_OUTPUT
	//Child objects
	
END_VAR

VAR_INPUT
		// Transfo
	IN_MesWarningTemp_IO				: BOOL ; 		// (NA) Warning Oil Temperature IO
	IN_MesAlarmTemp_IO					: BOOL ; 		// (NA) Alarm Oil Temperature   IO
	IN_MesAlarmGas_IO					: BOOL ; 		// (NA) Gas Alarm               IO
	IN_MesAlarmPressure_IO				: BOOL ; 		// (NA) Oil Pressure Alarm		IO
	IN_MesAlarmsSynthesis_IO			: BOOL ;        // (NA) Alarms synthesis        IO 
	
END_VAR

VAR
MesDataExd					: Transfo_MV ; 
	Emul_Alarm_Temp						: BOOL := FALSE;			
	Emul_Alarm_Synthesis				: BOOL := FALSE;
	
END_VAR

METHOD M_Execute
//////////////////
//  Method Calls 
/////////////////

VAR 
	// Method local variables (reinitialized at each cycle) 
	
END_VAR
 MesDataExd.MesData.MesAlarmTemp 			:= Emul_Alarm_Temp;			
MesDataExd.MesData.MesAlarmsSynthesis 		:= Emul_Alarm_Synthesis;
END_METHOD

END_FUNCTION_BLOCK

// ---- 01_Equipement_Library/Transfo/FB_Transfo_MVCom.TcPOU
FUNCTION_BLOCK FB_Transfo_MVCom EXTENDS FB_Transfo_Base

//////////////////
// High Voltage transformer with Transfo or DMCR detection . 
//////////////////

VAR_INPUT PERSISTENT
	// Parameters of the Object (instance/model specific) 
	
END_VAR

VAR_OUTPUT
	//Child objects
	
END_VAR

VAR_INPUT

	
END_VAR

VAR
MesDataExd					: Transfo_MV ; 
		
END_VAR

END_FUNCTION_BLOCK

// ---- 01_Equipement_Library/UPS/FB_UPS_Base.TcPOU
FUNCTION_BLOCK FB_UPS_Base
//////////////////
// UPS 
//////////////////
VAR_INPUT PERSISTENT
	// Parameters of the Object (instance/model specific) 
		ParamTimeOut				: TIME := T#2S;		//  (s)Modbus Timeout
		ParamClockReadTime			: TIME := T#1S;		// (s) Modbus Reading Frequency 
		ParamNC						: BOOL :=FALSE ; 	// False: TRUE = Closed , True : TRUE = opened

		
		ParamTempoComAlarm			: TIME := T#2S;		// (s)Tempo before raising a communication alarm
		ParamTempoComWarning		: TIME := T#1S;		// (s)Tempo before raising a communication warning
		ParamEBatt  				: REAL := 225; 		// (Wh) Emulateur : Ebat for 48V
END_VAR

VAR_OUTPUT
	//Child objects
		OUT_CmdRelance_IO			: BOOL;
END_VAR

VAR_INPUT
	// I/O Inputs
		IN_MesDischarging_IO		: BOOL;
		IN_MesBatLow_IO		   		: BOOL;
		IN_MesFault_IO				: BOOL;

		IN_CmdRelanceChargeur_IO	: BOOL;
		
		IN_CmdToggleRead			: BOOL;
		IN_CmdReset_L				: BOOL ; 
END_VAR

VAR
	//M_ALARMMANAGEMENT VARIABLES//
		TON_ComAlarm				: TON;
		TON_ComWarning				: TON;	

		MesWarningCom				: BOOL ; 			// (NA) [P,H] True if bad modbus communication 
			
	//M_READ//
//	MesDataExd					: UPS ; 

	//M_EXECUTE //
		TP1							: TP;

		ClockRead		AT %Q*		: BOOL;

		   		
    //M_CP VARIABLES//
		Trig_Cmd_Read				: R_TRIG;                                                                                        
                                                                                       
		CmdRelanceChargeur			: BOOL;
		CP_Relance					: BOOL;
		TP_Relance					: TP;
		ParamTP_Impulsion			: TIME:=T#5S;

	// EMULATOR //
	
		
END_VAR

METHOD M_Execute
//////////////////
//  Method Calls 
/////////////////

VAR 
	// Method local variables (reinitialized at each cycle) 

END_VAR
END_METHOD

END_FUNCTION_BLOCK

// ---- 01_Equipement_Library/UPS/FB_UPS_CXC.TcPOU
FUNCTION_BLOCK FB_UPS_CXC EXTENDS FB_UPS_Base
//////////////////
// UPS 
//////////////////
VAR_INPUT PERSISTENT
	// Parameters of the Object (instance/model specific) 

		ParamIPAddress				: STRING 	:= '192.168.20.66'; 	// (NA)Config: IP Adress of PV INverter
		ParamUnitID 				: BYTE  	:= 1; 			  		// (NA)   Modbus Unit ID. 
		ParamTCPPort				: UINT		:= 502;					// (NA) TCP port for modbus
		
END_VAR

VAR_OUTPUT
	//Child objects
	
END_VAR

VAR_INPUT
	// I/O Inputs
		IN_MesCbUPS_IO				: BOOL ; // 1 = opened. 
END_VAR

VAR
	//M_ALARMMANAGEMENT VARIABLES//

	//M_READ//
		MesDataExd						AT %Q*	: UPS_CXC ; 
		AX_ModbusRead		   		: ARRAY [1..2] OF FB_ModbusRead ; 					// (NA) FB for Modbus Reading
		ModbusReadInput				: FB_ModbusReadInput ; 		       
                                 
		MesBlock_Temp 				: ARRAY [1..2] OF ARRAY[1..120]  OF WORD; 			// (NA) Temporary Block with multiple modbus reading (Caution : Double Word variables)
		MesBlockInput				: ARRAY[1..1] OF BYTE ; 
		
	
	//M_EXECUTE //
		bInit: BOOL;
		
END_VAR

METHOD M_Execute
//////////////////
//  Method Calls 
/////////////////

VAR 
	// Method local variables (reinitialized at each cycle) 

END_VAR

IF bInit THEN
	bInit := FALSE ; 
MesDataExd.MesData.MesSoC := 50 ; 
END_IF

MesDataExd.MesIdc := 3 ; 

MesDataExd.MesUBatt := 47.5 ; 
IF MesDataExd.MesData.MesSoC >=100 THEN 
MesDataExd.MesData.MesIBatt := SEL(A1_SUBMV.A1_MainMVCB.MesDataExd.MesData.MesClosed , MesDataExd.MesData.MesIdc ,0   ) ; // can only be negative discharging 
ELSE
MesDataExd.MesData.MesIBatt :=  SEL(A1_SUBMV.A1_MainMVCB.MesDataExd.MesData.MesClosed , MesDataExd.MesData.MesIdc , 4   ) ;
END_IF
MesDataExd.MesSoC :=  MAX( 0 , MesDataExd.MesData.MesSoC  + 100.MesDataExd.MesData.MesIBatt*.MesDataExd.MesData.MesUBatt * 1/3600000 * ParamCycleTime_Emul / ParamEBatt ) ; 


MesDataExd.MesIload  := MesDataExd.MesData.MesIdc + MesDataExd.MesData.MesIBatt ; 

MesDataExd.MesUdc :=  SEL(A1_SUBMV.MesDataExd.MesData.A1_MainMVCB.MesDataExd.MesData.MesClosed  MesDataExd.MesData.MesUBatt , 48 ) ;; 
MesDataExd.MesUac	:= SEL(A1_SUBMV.MesDataExd.MesData.A1_MainMVCB.MesDataExd.MesData.MesClosed  ,0 , 230 ) ;

MesDataExd.MesData.MesBatteryLow := MesDataExd.MesData.MesSoC < 20 ; // Low battery capacity 
MesDataExd.MesData.MesDischarging := MesDataExd.MesData.MesIBatt < 0; 
MesDataExd.MesData.MesFaultSynthesis := MesDataExd.MesData.MesBatteryLow OR MesDataExd.MesData.MesDischarging ;
END_METHOD

END_FUNCTION_BLOCK

// ---- 01_Equipement_Library/UPS/FB_UPS_Eneris.TcPOU
FUNCTION_BLOCK FB_UPS_ENERIS EXTENDS FB_UPS_Base
//////////////////
// UPS 
//////////////////
VAR_INPUT PERSISTENT
	// Parameters of the Object (instance/model specific) 
	
END_VAR

VAR_OUTPUT
	//Child objects
	
END_VAR

VAR_INPUT
	// I/O Inputs
		IN_MesCbUPS_IO					: BOOL ; // 1 = opened. 
END_VAR

VAR
	//M_ALARMMANAGEMENT VARIABLES//
		
	//M_READ//

	MesDataExd				: UPS_ENERIS ; 
	
		
	//M_EXECUTE //
		
	
END_VAR

METHOD M_Execute
//////////////////
//  Method Calls 
/////////////////

VAR 
	// Method local variables (reinitialized at each cycle) 

END_VAR
END_METHOD

END_FUNCTION_BLOCK

// ---- 01_Equipement_Library/UPS/FB_UPS_PS10048.TcPOU
FUNCTION_BLOCK FB_UPS_PS10048 EXTENDS FB_UPS_Base
//////////////////
// SEPAM system for High Voltage or Low Voltage Grid Protection. 
//////////////////

VAR_INPUT 
	ParamTcpPort				: UINT:=502;
	ParamIPAddress				: STRING; 
	ParamUnitID					: BYTE; 
END_VAR

VAR_OUTPUT
	
END_VAR

VAR_INPUT

END_VAR

VAR
MesDataExd    	AT %Q*	: UPS_PS10048;
	FB_ModbusRead	          	: ARRAY[1..4] OF FB_ModbusRead; 
			
	MesBlock1_Temp 				: ARRAY [1..1] OF WORD; 
	MesBlock2_Temp 				: ARRAY [1..11] OF WORD; 
	MesBlock3_Temp 				: ARRAY [1..8] OF WORD; 
	MesBlock4_Temp 				: ARRAY [1..2] OF WORD; 
	
	AX_ModbusReadAlarm			: ARRAY[1..4] OF BOOL;
	AX_ModbusReadAlarmId		: ARRAY[1..4] OF UDINT;	
	
	//M_EXECUTE //
	bInit: BOOL;
	
	
	// Emulator 
	Emul_MesAlamCom 			: BOOL := FALSE;
	Emul_MesAlarm_AcLow			: BOOL := FALSE;
	Emul_MesAlarm_AcOff			: BOOL := FALSE;
	Emul_MesAlarm_Charger		: BOOL := FALSE;
	
END_VAR

METHOD M_Execute
//////////////////
//  Method Calls 
/////////////////

VAR_INPUT
	
END_VAR
VAR 
	MW					: FB_MergeWordsToFloat;
	MW_1				: FB_MergeWordsToDint;
END_VAR
	//COM
MesDataExd.MesData.MesAlarmCom 	:= Emul_MesAlamCom;
MesDataExd.MesData.MesCapacity_Nom 		:= ParamEBatt.MesDataExd.MesData.MesUdc_48V; 	
	
MesDataExd.MesData.MesUdc_12V 			:= 12;		 

MesDataExd.MesData.MesCapacity_Nom 		:= 37000;
	                                
    MesDataExd.MesData.MesAlarm_AcLow		:= Emul_MesAlarm_AcLow;
	 
IF bInit THEN
	bInit 				:= FALSE; 
MesDataExd.MesData.MesSoC 	:= 50; 
END_IF

MesDataExd.MesUBatt 	:= 47.5 ; 
IF MesDataExd.MesData.MesSoC 	>=100 THEN 
MesDataExd.MesData.MesIdc_Bat  := SEL(A1_SUBMV.A1_MainMVCB.MesDataExd.MesData.MesClosed , -.MesDataExd.MesData.MesIdc_12V , 0) ; 			// can only be negative discharging 
ELSE
MesDataExd.MesData.MesIdc_Bat :=  SEL(A1_SUBMV.A1_MainMVCB.MesDataExd.MesData.MesClosed , MesDataExd.MesData.MesIdc_12V , 4) ;
END_IF

MesDataExd.MesSoC	  				:=  MAX( 0, MesDataExd.MesData.MesSoC  + 100.MesDataExd.MesData.MesIdc_Bat*.MesDataExd.MesData.MesUBatt * 1/3600000 * ParamCycleTime_Emul / ParamEBatt); 
MesDataExd.MesUdc_48V 				:=  SEL(A1_SUBMV.A1_MainMVCB.MesDataExd.MesData.MesClosed, MesDataExd.MesData.MesUBatt, 48) ; 

MesDataExd.MesData.MesAlarm_Ulow  	:= MesDataExd.MesData.MesSoC < 20 ; // Low battery capacity 
MesDataExd.MesData.MesDischarging 	:= MesDataExd.MesData.MesIdc_Bat < 0; 
	
MesDataExd.MesAlarm_AcOff 			:= Emul_MesAlarm_AcOff;
MesDataExd.MesAlarm_AcLow 			:= Emul_MesAlarm_AcLow;
MesDataExd.MesFault_Charger			:= Emul_MesAlarm_Charger;

MesdataExd.MesFault_Minor   		:= MesDataExd.MesData.MesAlarm_AcLow OR MesDataExd.MesData.MesAlarm_Ulow ;
MesdataExd.MesFault_Major   		:= MesDataExd.MesData.MesSoC < 10 OR MesDataExd.MesData.MesAlarm_AcOff OR MesDataExd.MesData.MesFault_Charger;
mesdataexd.MesAlarm_GeneralOff		:= MesDataExd.MesData.MesAlarm_AcOff OR MesDataExd.MesData.MesSoC < 5;
END_METHOD

END_FUNCTION_BLOCK

// ---- 04_Application/ADS/ADS_Param.TcPOU
PROGRAM ADS_Param
VAR
END_VAR

SignalName[1]:='GVL_CFG.AX_PTR[1].A1_INV_Smartlogger.MesDataExd.MesData.;	bClockIO[1]:=FALSE;	Taille[1]:=SIZEOF(GVL_CFG.AX_PTR[1].A1_INV_Smartlogger.MesDataExd.MesData.;	Address[1]:=ADR(GVL_CFG.AX_PTR[1].A1_INV_Smartlogger.MesDataExd.MesData.;	ReadAdsType[1]:=FALSE;	WriteAdsType[1]:=TRUE;
SignalName[2]:='GVL_CFG.AX_PTR[2].A1_INV_Smartlogger.MesDataExd.MesData.;	bClockIO[2]:=FALSE;	Taille[2]:=SIZEOF(GVL_CFG.AX_PTR[2].A1_INV_Smartlogger.MesDataExd.MesData.;	Address[2]:=ADR(GVL_CFG.AX_PTR[2].A1_INV_Smartlogger.MesDataExd.MesData.;	ReadAdsType[2]:=FALSE;	WriteAdsType[2]:=TRUE;
SignalName[3]:='GVL_CFG.AX_PTR[3].A1_INV_Smartlogger.MesDataExd.MesData.;	bClockIO[3]:=FALSE;	Taille[3]:=SIZEOF(GVL_CFG.AX_PTR[3].A1_INV_Smartlogger.MesDataExd.MesData.;	Address[3]:=ADR(GVL_CFG.AX_PTR[3].A1_INV_Smartlogger.MesDataExd.MesData.;	ReadAdsType[3]:=FALSE;	WriteAdsType[3]:=TRUE;
SignalName[4]:='GVL_CFG.AX_PTR[4].A1_INV_Smartlogger.MesDataExd.MesData.;	bClockIO[4]:=FALSE;	Taille[4]:=SIZEOF(GVL_CFG.AX_PTR[4].A1_INV_Smartlogger.MesDataExd.MesData.;	Address[4]:=ADR(GVL_CFG.AX_PTR[4].A1_INV_Smartlogger.MesDataExd.MesData.;	ReadAdsType[4]:=FALSE;	WriteAdsType[4]:=TRUE;
SignalName[5]:='GVL_CFG.AX_PTR[1].A1_INV_Smartlogger.WriteBlock_Temp';	bClockIO[5]:=TRUE;	Taille[5]:=SIZEOF(GVL_CFG.AX_PTR[1].A1_INV_Smartlogger.WriteBlock_Temp);	Address[5]:=ADR(GVL_CFG.AX_PTR[1].A1_INV_Smartlogger.WriteBlock_Temp);	ReadAdsType[5]:=TRUE;	WriteAdsType[5]:=FALSE;
SignalName[6]:='GVL_CFG.AX_PTR[2].A1_INV_Smartlogger.WriteBlock_Temp';	bClockIO[6]:=TRUE;	Taille[6]:=SIZEOF(GVL_CFG.AX_PTR[2].A1_INV_Smartlogger.WriteBlock_Temp);	Address[6]:=ADR(GVL_CFG.AX_PTR[2].A1_INV_Smartlogger.WriteBlock_Temp);	ReadAdsType[6]:=TRUE;	WriteAdsType[6]:=FALSE;
SignalName[7]:='GVL_CFG.AX_PTR[3].A1_INV_Smartlogger.WriteBlock_Temp';	bClockIO[7]:=TRUE;	Taille[7]:=SIZEOF(GVL_CFG.AX_PTR[3].A1_INV_Smartlogger.WriteBlock_Temp);	Address[7]:=ADR(GVL_CFG.AX_PTR[3].A1_INV_Smartlogger.WriteBlock_Temp);	ReadAdsType[7]:=TRUE;	WriteAdsType[7]:=FALSE;
SignalName[8]:='GVL_CFG.AX_PTR[4].A1_INV_Smartlogger.WriteBlock_Temp';	bClockIO[8]:=TRUE;	Taille[8]:=SIZEOF(GVL_CFG.AX_PTR[4].A1_INV_Smartlogger.WriteBlock_Temp);	Address[8]:=ADR(GVL_CFG.AX_PTR[4].A1_INV_Smartlogger.WriteBlock_Temp);	ReadAdsType[8]:=TRUE;	WriteAdsType[8]:=FALSE;
SignalName[9]:='GVL_CFG.AX_PTR[1].A1_INV_Smartlogger.ClockRead';	bClockIO[9]:=TRUE;	Taille[9]:=SIZEOF(GVL_CFG.AX_PTR[1].A1_INV_Smartlogger.ClockRead);	Address[9]:=ADR(GVL_CFG.AX_PTR[1].A1_INV_Smartlogger.ClockRead);	ReadAdsType[9]:=TRUE;	WriteAdsType[9]:=FALSE;
SignalName[10]:='GVL_CFG.AX_PTR[2].A1_INV_Smartlogger.ClockRead';	bClockIO[10]:=TRUE;	Taille[10]:=SIZEOF(GVL_CFG.AX_PTR[2].A1_INV_Smartlogger.ClockRead);	Address[10]:=ADR(GVL_CFG.AX_PTR[2].A1_INV_Smartlogger.ClockRead);	ReadAdsType[10]:=TRUE;	WriteAdsType[10]:=FALSE;
SignalName[11]:='GVL_CFG.AX_PTR[3].A1_INV_Smartlogger.ClockRead';	bClockIO[11]:=TRUE;	Taille[11]:=SIZEOF(GVL_CFG.AX_PTR[3].A1_INV_Smartlogger.ClockRead);	Address[11]:=ADR(GVL_CFG.AX_PTR[3].A1_INV_Smartlogger.ClockRead);	ReadAdsType[11]:=TRUE;	WriteAdsType[11]:=FALSE;
SignalName[12]:='GVL_CFG.AX_PTR[4].A1_INV_Smartlogger.ClockRead';	bClockIO[12]:=TRUE;	Taille[12]:=SIZEOF(GVL_CFG.AX_PTR[4].A1_INV_Smartlogger.ClockRead);	Address[12]:=ADR(GVL_CFG.AX_PTR[4].A1_INV_Smartlogger.ClockRead);	ReadAdsType[12]:=TRUE;	WriteAdsType[12]:=FALSE;
SignalName[13]:='GVL_CFG.AX_PTR[1].A1_INV_Smartlogger.ClockWrite';	bClockIO[13]:=TRUE;	Taille[13]:=SIZEOF(GVL_CFG.AX_PTR[1].A1_INV_Smartlogger.ClockWrite);	Address[13]:=ADR(GVL_CFG.AX_PTR[1].A1_INV_Smartlogger.ClockWrite);	ReadAdsType[13]:=TRUE;	WriteAdsType[13]:=FALSE;
SignalName[14]:='GVL_CFG.AX_PTR[2].A1_INV_Smartlogger.ClockWrite';	bClockIO[14]:=TRUE;	Taille[14]:=SIZEOF(GVL_CFG.AX_PTR[2].A1_INV_Smartlogger.ClockWrite);	Address[14]:=ADR(GVL_CFG.AX_PTR[2].A1_INV_Smartlogger.ClockWrite);	ReadAdsType[14]:=TRUE;	WriteAdsType[14]:=FALSE;
SignalName[15]:='GVL_CFG.AX_PTR[3].A1_INV_Smartlogger.ClockWrite';	bClockIO[15]:=TRUE;	Taille[15]:=SIZEOF(GVL_CFG.AX_PTR[3].A1_INV_Smartlogger.ClockWrite);	Address[15]:=ADR(GVL_CFG.AX_PTR[3].A1_INV_Smartlogger.ClockWrite);	ReadAdsType[15]:=TRUE;	WriteAdsType[15]:=FALSE;
SignalName[16]:='GVL_CFG.AX_PTR[4].A1_INV_Smartlogger.ClockWrite';	bClockIO[16]:=TRUE;	Taille[16]:=SIZEOF(GVL_CFG.AX_PTR[4].A1_INV_Smartlogger.ClockWrite);	Address[16]:=ADR(GVL_CFG.AX_PTR[4].A1_INV_Smartlogger.ClockWrite);	ReadAdsType[16]:=TRUE;	WriteAdsType[16]:=FALSE;
SignalName[17]:='GVL_CFG.AX_PTR[1].AX_INV[1].MesDataExd.MesData.;	bClockIO[17]:=FALSE;	Taille[17]:=SIZEOF(GVL_CFG.AX_PTR[1].AX_INV[1].MesDataExd.MesData.;	Address[17]:=ADR(GVL_CFG.AX_PTR[1].AX_INV[1].MesDataExd.MesData.;	ReadAdsType[17]:=FALSE;	WriteAdsType[17]:=TRUE;
SignalName[18]:='GVL_CFG.AX_PTR[1].AX_INV[2].MesDataExd.MesData.;	bClockIO[18]:=FALSE;	Taille[18]:=SIZEOF(GVL_CFG.AX_PTR[1].AX_INV[2].MesDataExd.MesData.;	Address[18]:=ADR(GVL_CFG.AX_PTR[1].AX_INV[2].MesDataExd.MesData.;	ReadAdsType[18]:=FALSE;	WriteAdsType[18]:=TRUE;
SignalName[19]:='GVL_CFG.AX_PTR[2].AX_INV[1].MesDataExd.MesData.;	bClockIO[19]:=FALSE;	Taille[19]:=SIZEOF(GVL_CFG.AX_PTR[2].AX_INV[1].MesDataExd.MesData.;	Address[19]:=ADR(GVL_CFG.AX_PTR[2].AX_INV[1].MesDataExd.MesData.;	ReadAdsType[19]:=FALSE;	WriteAdsType[19]:=TRUE;
SignalName[20]:='GVL_CFG.AX_PTR[2].AX_INV[2].MesDataExd.MesData.;	bClockIO[20]:=FALSE;	Taille[20]:=SIZEOF(GVL_CFG.AX_PTR[2].AX_INV[2].MesDataExd.MesData.;	Address[20]:=ADR(GVL_CFG.AX_PTR[2].AX_INV[2].MesDataExd.MesData.;	ReadAdsType[20]:=FALSE;	WriteAdsType[20]:=TRUE;
SignalName[21]:='GVL_CFG.AX_PTR[3].AX_INV[1].MesDataExd.MesData.;	bClockIO[21]:=FALSE;	Taille[21]:=SIZEOF(GVL_CFG.AX_PTR[3].AX_INV[1].MesDataExd.MesData.;	Address[21]:=ADR(GVL_CFG.AX_PTR[3].AX_INV[1].MesDataExd.MesData.;	ReadAdsType[21]:=FALSE;	WriteAdsType[21]:=TRUE;
SignalName[22]:='GVL_CFG.AX_PTR[3].AX_INV[2].MesDataExd.MesData.;	bClockIO[22]:=FALSE;	Taille[22]:=SIZEOF(GVL_CFG.AX_PTR[3].AX_INV[2].MesDataExd.MesData.;	Address[22]:=ADR(GVL_CFG.AX_PTR[3].AX_INV[2].MesDataExd.MesData.;	ReadAdsType[22]:=FALSE;	WriteAdsType[22]:=TRUE;
SignalName[23]:='GVL_CFG.AX_PTR[4].AX_INV[1].MesDataExd.MesData.;	bClockIO[23]:=FALSE;	Taille[23]:=SIZEOF(GVL_CFG.AX_PTR[4].AX_INV[1].MesDataExd.MesData.;	Address[23]:=ADR(GVL_CFG.AX_PTR[4].AX_INV[1].MesDataExd.MesData.;	ReadAdsType[23]:=FALSE;	WriteAdsType[23]:=TRUE;
SignalName[24]:='GVL_CFG.AX_PTR[4].AX_INV[2].MesDataExd.MesData.;	bClockIO[24]:=FALSE;	Taille[24]:=SIZEOF(GVL_CFG.AX_PTR[4].AX_INV[2].MesDataExd.MesData.;	Address[24]:=ADR(GVL_CFG.AX_PTR[4].AX_INV[2].MesDataExd.MesData.;	ReadAdsType[24]:=FALSE;	WriteAdsType[24]:=TRUE;
SignalName[25]:='GVL_CFG.AX_PTR[1].AX_INV[1].ClockRead';	bClockIO[25]:=TRUE;	Taille[25]:=SIZEOF(GVL_CFG.AX_PTR[1].AX_INV[1].ClockRead);	Address[25]:=ADR(GVL_CFG.AX_PTR[1].AX_INV[1].ClockRead);	ReadAdsType[25]:=TRUE;	WriteAdsType[25]:=FALSE;
SignalName[26]:='GVL_CFG.AX_PTR[1].AX_INV[2].ClockRead';	bClockIO[26]:=TRUE;	Taille[26]:=SIZEOF(GVL_CFG.AX_PTR[1].AX_INV[2].ClockRead);	Address[26]:=ADR(GVL_CFG.AX_PTR[1].AX_INV[2].ClockRead);	ReadAdsType[26]:=TRUE;	WriteAdsType[26]:=FALSE;
SignalName[27]:='GVL_CFG.AX_PTR[2].AX_INV[1].ClockRead';	bClockIO[27]:=TRUE;	Taille[27]:=SIZEOF(GVL_CFG.AX_PTR[2].AX_INV[1].ClockRead);	Address[27]:=ADR(GVL_CFG.AX_PTR[2].AX_INV[1].ClockRead);	ReadAdsType[27]:=TRUE;	WriteAdsType[27]:=FALSE;
SignalName[28]:='GVL_CFG.AX_PTR[2].AX_INV[2].ClockRead';	bClockIO[28]:=TRUE;	Taille[28]:=SIZEOF(GVL_CFG.AX_PTR[2].AX_INV[2].ClockRead);	Address[28]:=ADR(GVL_CFG.AX_PTR[2].AX_INV[2].ClockRead);	ReadAdsType[28]:=TRUE;	WriteAdsType[28]:=FALSE;
SignalName[29]:='GVL_CFG.AX_PTR[3].AX_INV[1].ClockRead';	bClockIO[29]:=TRUE;	Taille[29]:=SIZEOF(GVL_CFG.AX_PTR[3].AX_INV[1].ClockRead);	Address[29]:=ADR(GVL_CFG.AX_PTR[3].AX_INV[1].ClockRead);	ReadAdsType[29]:=TRUE;	WriteAdsType[29]:=FALSE;
SignalName[30]:='GVL_CFG.AX_PTR[3].AX_INV[2].ClockRead';	bClockIO[30]:=TRUE;	Taille[30]:=SIZEOF(GVL_CFG.AX_PTR[3].AX_INV[2].ClockRead);	Address[30]:=ADR(GVL_CFG.AX_PTR[3].AX_INV[2].ClockRead);	ReadAdsType[30]:=TRUE;	WriteAdsType[30]:=FALSE;
SignalName[31]:='GVL_CFG.AX_PTR[4].AX_INV[1].ClockRead';	bClockIO[31]:=TRUE;	Taille[31]:=SIZEOF(GVL_CFG.AX_PTR[4].AX_INV[1].ClockRead);	Address[31]:=ADR(GVL_CFG.AX_PTR[4].AX_INV[1].ClockRead);	ReadAdsType[31]:=TRUE;	WriteAdsType[31]:=FALSE;
SignalName[32]:='GVL_CFG.AX_PTR[4].AX_INV[2].ClockRead';	bClockIO[32]:=TRUE;	Taille[32]:=SIZEOF(GVL_CFG.AX_PTR[4].AX_INV[2].ClockRead);	Address[32]:=ADR(GVL_CFG.AX_PTR[4].AX_INV[2].ClockRead);	ReadAdsType[32]:=TRUE;	WriteAdsType[32]:=FALSE;
SignalName[33]:='GVL_CFG.AX_PTR[1].AX_INV[1].ClockWrite';	bClockIO[33]:=TRUE;	Taille[33]:=SIZEOF(GVL_CFG.AX_PTR[1].AX_INV[1].ClockWrite);	Address[33]:=ADR(GVL_CFG.AX_PTR[1].AX_INV[1].ClockWrite);	ReadAdsType[33]:=TRUE;	WriteAdsType[33]:=FALSE;
SignalName[34]:='GVL_CFG.AX_PTR[1].AX_INV[2].ClockWrite';	bClockIO[34]:=TRUE;	Taille[34]:=SIZEOF(GVL_CFG.AX_PTR[1].AX_INV[2].ClockWrite);	Address[34]:=ADR(GVL_CFG.AX_PTR[1].AX_INV[2].ClockWrite);	ReadAdsType[34]:=TRUE;	WriteAdsType[34]:=FALSE;
SignalName[35]:='GVL_CFG.AX_PTR[2].AX_INV[1].ClockWrite';	bClockIO[35]:=TRUE;	Taille[35]:=SIZEOF(GVL_CFG.AX_PTR[2].AX_INV[1].ClockWrite);	Address[35]:=ADR(GVL_CFG.AX_PTR[2].AX_INV[1].ClockWrite);	ReadAdsType[35]:=TRUE;	WriteAdsType[35]:=FALSE;
SignalName[36]:='GVL_CFG.AX_PTR[2].AX_INV[2].ClockWrite';	bClockIO[36]:=TRUE;	Taille[36]:=SIZEOF(GVL_CFG.AX_PTR[2].AX_INV[2].ClockWrite);	Address[36]:=ADR(GVL_CFG.AX_PTR[2].AX_INV[2].ClockWrite);	ReadAdsType[36]:=TRUE;	WriteAdsType[36]:=FALSE;
SignalName[37]:='GVL_CFG.AX_PTR[3].AX_INV[1].ClockWrite';	bClockIO[37]:=TRUE;	Taille[37]:=SIZEOF(GVL_CFG.AX_PTR[3].AX_INV[1].ClockWrite);	Address[37]:=ADR(GVL_CFG.AX_PTR[3].AX_INV[1].ClockWrite);	ReadAdsType[37]:=TRUE;	WriteAdsType[37]:=FALSE;
SignalName[38]:='GVL_CFG.AX_PTR[3].AX_INV[2].ClockWrite';	bClockIO[38]:=TRUE;	Taille[38]:=SIZEOF(GVL_CFG.AX_PTR[3].AX_INV[2].ClockWrite);	Address[38]:=ADR(GVL_CFG.AX_PTR[3].AX_INV[2].ClockWrite);	ReadAdsType[38]:=TRUE;	WriteAdsType[38]:=FALSE;
SignalName[39]:='GVL_CFG.AX_PTR[4].AX_INV[1].ClockWrite';	bClockIO[39]:=TRUE;	Taille[39]:=SIZEOF(GVL_CFG.AX_PTR[4].AX_INV[1].ClockWrite);	Address[39]:=ADR(GVL_CFG.AX_PTR[4].AX_INV[1].ClockWrite);	ReadAdsType[39]:=TRUE;	WriteAdsType[39]:=FALSE;
SignalName[40]:='GVL_CFG.AX_PTR[4].AX_INV[2].ClockWrite';	bClockIO[40]:=TRUE;	Taille[40]:=SIZEOF(GVL_CFG.AX_PTR[4].AX_INV[2].ClockWrite);	Address[40]:=ADR(GVL_CFG.AX_PTR[4].AX_INV[2].ClockWrite);	ReadAdsType[40]:=TRUE;	WriteAdsType[40]:=FALSE;
SignalName[41]:='GVL_CFG.A1_SUBMV.A1_ProtectRelay.MesDataExd.MesData.;	bClockIO[41]:=FALSE;	Taille[41]:=SIZEOF(GVL_CFG.A1_SUBMV.A1_ProtectRelay.MesDataExd.MesData.;	Address[41]:=ADR(GVL_CFG.A1_SUBMV.A1_ProtectRelay.MesDataExd.MesData.;	ReadAdsType[41]:=FALSE;	WriteAdsType[41]:=TRUE;
SignalName[42]:='GVL_CFG.A1_SUBMV.A1_ProtectRelay.ClockRead';	bClockIO[42]:=TRUE;	Taille[42]:=SIZEOF(GVL_CFG.A1_SUBMV.A1_ProtectRelay.ClockRead);	Address[42]:=ADR(GVL_CFG.A1_SUBMV.A1_ProtectRelay.ClockRead);	ReadAdsType[42]:=TRUE;	WriteAdsType[42]:=FALSE;
SignalName[43]:='GVL_CFG.A1_SUBMV.A1_PM.MesDataExd.MesData.;	bClockIO[43]:=FALSE;	Taille[43]:=SIZEOF(GVL_CFG.A1_SUBMV.A1_PM.MesDataExd.MesData.;	Address[43]:=ADR(GVL_CFG.A1_SUBMV.A1_PM.MesDataExd.MesData.;	ReadAdsType[43]:=FALSE;	WriteAdsType[43]:=TRUE;
SignalName[44]:='GVL_CFG.A1_SUBMV.A1_PM.ClockRead';	bClockIO[44]:=TRUE;	Taille[44]:=SIZEOF(GVL_CFG.A1_SUBMV.A1_PM.ClockRead);	Address[44]:=ADR(GVL_CFG.A1_SUBMV.A1_PM.ClockRead);	ReadAdsType[44]:=TRUE;	WriteAdsType[44]:=FALSE;
SignalName[45]:='GVL_CFG.A1_SUBMV.A1_PM_Aux.MesDataExd.MesData.;	bClockIO[45]:=FALSE;	Taille[45]:=SIZEOF(GVL_CFG.A1_SUBMV.A1_PM_Aux.MesDataExd.MesData.;	Address[45]:=ADR(GVL_CFG.A1_SUBMV.A1_PM_Aux.MesDataExd.MesData.;	ReadAdsType[45]:=FALSE;	WriteAdsType[45]:=TRUE;
SignalName[46]:='GVL_CFG.A1_SUBMV.A1_PM_Aux.ClockRead';	bClockIO[46]:=TRUE;	Taille[46]:=SIZEOF(GVL_CFG.A1_SUBMV.A1_PM_Aux.ClockRead);	Address[46]:=ADR(GVL_CFG.A1_SUBMV.A1_PM_Aux.ClockRead);	ReadAdsType[46]:=TRUE;	WriteAdsType[46]:=FALSE;
SignalName[47]:='GVL_CFG.A1_SUBMV.A1_UPS_48v.ClockRead';	bClockIO[47]:=TRUE;	Taille[47]:=SIZEOF(GVL_CFG.A1_SUBMV.A1_UPS_48v.ClockRead);	Address[47]:=ADR(GVL_CFG.A1_SUBMV.A1_UPS_48v.ClockRead);	ReadAdsType[47]:=TRUE;	WriteAdsType[47]:=FALSE;
SignalName[48]:='GVL_CFG.A1_SUBMV.A1_UPS_24v.ClockRead';	bClockIO[48]:=TRUE;	Taille[48]:=SIZEOF(GVL_CFG.A1_SUBMV.A1_UPS_24v.ClockRead);	Address[48]:=ADR(GVL_CFG.A1_SUBMV.A1_UPS_24v.ClockRead);	ReadAdsType[48]:=TRUE;	WriteAdsType[48]:=FALSE;
SignalName[49]:='PRG_IO.MesCouplerStateSUBMV';	bClockIO[49]:=TRUE;	Taille[49]:=SIZEOF(PRG_IO.MesCouplerStateSUBMV);	Address[49]:=ADR(PRG_IO.MesCouplerStateSUBMV);	ReadAdsType[49]:=FALSE;	WriteAdsType[49]:=TRUE;
SignalName[50]:='PRG_IO.MesIO_SUBMV_EL1809_1';	bClockIO[50]:=TRUE;	Taille[50]:=SIZEOF(PRG_IO.MesIO_SUBMV_EL1809_1);	Address[50]:=ADR(PRG_IO.MesIO_SUBMV_EL1809_1);	ReadAdsType[50]:=FALSE;	WriteAdsType[50]:=TRUE;
SignalName[51]:='PRG_IO.MesIO_SUBMV_EL1809_2';	bClockIO[51]:=TRUE;	Taille[51]:=SIZEOF(PRG_IO.MesIO_SUBMV_EL1809_2);	Address[51]:=ADR(PRG_IO.MesIO_SUBMV_EL1809_2);	ReadAdsType[51]:=FALSE;	WriteAdsType[51]:=TRUE;
SignalName[52]:='PRG_IO.MesIO_SUBMV_EL1809_3';	bClockIO[52]:=TRUE;	Taille[52]:=SIZEOF(PRG_IO.MesIO_SUBMV_EL1809_3);	Address[52]:=ADR(PRG_IO.MesIO_SUBMV_EL1809_3);	ReadAdsType[52]:=FALSE;	WriteAdsType[52]:=TRUE;
SignalName[53]:='PRG_IO.MesIO_SUBMV_EL2809_4';	bClockIO[53]:=TRUE;	Taille[53]:=SIZEOF(PRG_IO.MesIO_SUBMV_EL2809_4);	Address[53]:=ADR(PRG_IO.MesIO_SUBMV_EL2809_4);	ReadAdsType[53]:=TRUE;	WriteAdsType[53]:=FALSE;
SignalName[54]:='PRG_IO.MesIO_SUBMV_EL3024_5';	bClockIO[54]:=TRUE;	Taille[54]:=SIZEOF(PRG_IO.MesIO_SUBMV_EL3024_5);	Address[54]:=ADR(PRG_IO.MesIO_SUBMV_EL3024_5);	ReadAdsType[54]:=FALSE;	WriteAdsType[54]:=TRUE;
SignalName[55]:='PRG_IO.MesIO_SUBMV_EL1809_14';	bClockIO[55]:=TRUE;	Taille[55]:=SIZEOF(PRG_IO.MesIO_SUBMV_EL1809_14);	Address[55]:=ADR(PRG_IO.MesIO_SUBMV_EL1809_14);	ReadAdsType[55]:=TRUE;	WriteAdsType[55]:=FALSE;
SignalName[56]:='PRG_IO.MesIO_PTR_1_EL3024_8';	bClockIO[56]:=TRUE;	Taille[56]:=SIZEOF(PRG_IO.MesIO_PTR_1_EL3024_8);	Address[56]:=ADR(PRG_IO.MesIO_PTR_1_EL3024_8);	ReadAdsType[56]:=FALSE;	WriteAdsType[56]:=TRUE;
SignalName[57]:='PRG_IO.MesIO_PTR_1_EL1809_9';	bClockIO[57]:=TRUE;	Taille[57]:=SIZEOF(PRG_IO.MesIO_PTR_1_EL1809_9);	Address[57]:=ADR(PRG_IO.MesIO_PTR_1_EL1809_9);	ReadAdsType[57]:=FALSE;	WriteAdsType[57]:=TRUE;
SignalName[58]:='PRG_IO.MesIO_PTR_1_EL2809_10';	bClockIO[58]:=TRUE;	Taille[58]:=SIZEOF(PRG_IO.MesIO_PTR_1_EL2809_10);	Address[58]:=ADR(PRG_IO.MesIO_PTR_1_EL2809_10);	ReadAdsType[58]:=TRUE;	WriteAdsType[58]:=FALSE;
SignalName[59]:='PRG_IO.MesIO_PTR_2_EL3024_8';	bClockIO[59]:=TRUE;	Taille[59]:=SIZEOF(PRG_IO.MesIO_PTR_2_EL3024_8);	Address[59]:=ADR(PRG_IO.MesIO_PTR_2_EL3024_8);	ReadAdsType[59]:=FALSE;	WriteAdsType[59]:=TRUE;
SignalName[60]:='PRG_IO.MesIO_PTR_2_EL1809_9';	bClockIO[60]:=TRUE;	Taille[60]:=SIZEOF(PRG_IO.MesIO_PTR_2_EL1809_9);	Address[60]:=ADR(PRG_IO.MesIO_PTR_2_EL1809_9);	ReadAdsType[60]:=FALSE;	WriteAdsType[60]:=TRUE;
SignalName[61]:='PRG_IO.MesIO_PTR_2_EL2809_10';	bClockIO[61]:=TRUE;	Taille[61]:=SIZEOF(PRG_IO.MesIO_PTR_2_EL2809_10);	Address[61]:=ADR(PRG_IO.MesIO_PTR_2_EL2809_10);	ReadAdsType[61]:=TRUE;	WriteAdsType[61]:=FALSE;
SignalName[62]:='PRG_IO.MesIO_PTR_3_EL3024_8';	bClockIO[62]:=TRUE;	Taille[62]:=SIZEOF(PRG_IO.MesIO_PTR_3_EL3024_8);	Address[62]:=ADR(PRG_IO.MesIO_PTR_3_EL3024_8);	ReadAdsType[62]:=FALSE;	WriteAdsType[62]:=TRUE;
SignalName[63]:='PRG_IO.MesIO_PTR_3_EL1809_9';	bClockIO[63]:=TRUE;	Taille[63]:=SIZEOF(PRG_IO.MesIO_PTR_3_EL1809_9);	Address[63]:=ADR(PRG_IO.MesIO_PTR_3_EL1809_9);	ReadAdsType[63]:=FALSE;	WriteAdsType[63]:=TRUE;
SignalName[64]:='PRG_IO.MesIO_PTR_3_EL2809_10';	bClockIO[64]:=TRUE;	Taille[64]:=SIZEOF(PRG_IO.MesIO_PTR_3_EL2809_10);	Address[64]:=ADR(PRG_IO.MesIO_PTR_3_EL2809_10);	ReadAdsType[64]:=TRUE;	WriteAdsType[64]:=FALSE;

END_PROGRAM

// ---- 04_Application/Checks/CheckBounds.TcPOU
// Code généré automatiquement : NE PAS MODIFIER
FUNCTION CheckBounds : DINT
VAR_INPUT
	index, lower, upper: DINT;
END_VAR

// Code généré automatiquement : Il s’agit d’une proposition d’implémentation.
{noflow}
Fault_Count_G(CU:=FALSE) ; 
IF  index < lower THEN
	CheckBounds := lower;
	Fault_Count_G(CU:=TRUE) ; 
ELSIF  index > upper THEN
	CheckBounds := upper;
	Fault_Count_G(CU:=TRUE) ; 
ELSE  
	CheckBounds := index;
END_IF
{flow}

END_FUNCTION

// ---- 04_Application/Checks/CheckDivDInt.TcPOU
// Code généré automatiquement : NE PAS MODIFIER
FUNCTION CheckDivDInt : DINT
VAR_INPUT
	divisor:DINT;
END_VAR

// Code généré automatiquement : Il s’agit d’une proposition d’implémentation.
{noflow}
IF divisor = 0 THEN
	CheckDivDInt:=1;
ELSE
	CheckDivDInt:=divisor;
END_IF;
{flow}

END_FUNCTION

// ---- 04_Application/Checks/CheckDivLInt.TcPOU
// Code généré automatiquement : NE PAS MODIFIER
FUNCTION CheckDivLInt : LINT
VAR_INPUT
	divisor:LINT;
END_VAR

// Code généré automatiquement : Il s’agit d’une proposition d’implémentation.
{noflow}
IF divisor = 0 THEN
	CheckDivLInt:=1;
ELSE
	CheckDivLInt:=divisor;
END_IF;
{flow}

END_FUNCTION

// ---- 04_Application/Checks/CheckDivLReal.TcPOU
// Code généré automatiquement : NE PAS MODIFIER
FUNCTION CheckDivLReal : LREAL
VAR_INPUT
	divisor:LREAL;
END_VAR

// Code généré automatiquement : Il s’agit d’une proposition d’implémentation.
{noflow}
IF divisor = 0 THEN
	CheckDivLReal:=1;
ELSE
	CheckDivLReal:=divisor;
END_IF;
{flow}

END_FUNCTION

// ---- 04_Application/Checks/CheckDivReal.TcPOU
// Code généré automatiquement : NE PAS MODIFIER
FUNCTION CheckDivReal : REAL
VAR_INPUT
	divisor:REAL;
END_VAR

// Code généré automatiquement : Il s’agit d’une proposition d’implémentation.
{noflow}
IF divisor = 0 THEN
	CheckDivReal:=1;
ELSE
	CheckDivReal:=divisor;
END_IF;
{flow}

END_FUNCTION

// ---- 04_Application/Checks/CheckLRangeSigned.TcPOU
// Code généré automatiquement : NE PAS MODIFIER
FUNCTION CheckLRangeSigned : LINT
VAR_INPUT
	value, lower, upper: LINT;
END_VAR

// Code généré automatiquement : Il s’agit d’une proposition d’implémentation.
{noflow}
IF (value < lower) THEN
	CheckLRangeSigned := lower;
ELSIF(value > upper) THEN
	CheckLRangeSigned := upper;
ELSE
	CheckLRangeSigned := value;
END_IF

{flow}

END_FUNCTION

// ---- 04_Application/Checks/CheckLRangeUnsigned.TcPOU
// Code généré automatiquement : NE PAS MODIFIER
FUNCTION CheckLRangeUnsigned : ULINT
VAR_INPUT
	value, lower, upper: ULINT;
END_VAR

// Code généré automatiquement : Il s’agit d’une proposition d’implémentation.
{noflow}
IF (value < lower) THEN
	CheckLRangeUnsigned := lower;
ELSIF(value > upper) THEN
	CheckLRangeUnsigned := upper;
ELSE
	CheckLRangeUnsigned := value;
END_IF
{flow}

END_FUNCTION

// ---- 04_Application/Checks/CheckPointer.TcPOU
// Code généré automatiquement : NE PAS MODIFIER
FUNCTION CheckPointer : POINTER TO BYTE
VAR_INPUT 
	ptToTest : POINTER TO BYTE; // Adresse de destination du pointeur
	iSize : DINT;		        // Taille du type indiqué par le pointeur.  (par exemple : 20 pour POINTER TO ARRAY [0..9] OF INT)
	iGran : DINT;		        // Granularité de l’accès au pointeur. Il s’agit de la taille du plus grand type de données non structuré dans le type indiqué par le pointeur.  (par exemple : 2 pour POINTER TO ARRAY [0..9] OF INT)
	bWrite: BOOL;		        // Indique l’accès en lecture ou en écriture. TRUE = accès en écriture.
END_VAR

// Code généré automatiquement : Il s’agit d’une proposition d’implémentation.
{noflow}
IF ptToTest=0 THEN
    ADSLOGSTR(ADSLOG_MSGTYPE_ERROR OR ADSLOG_MSGTYPE_STRING,'CheckPointer failed due to invalid address.','');
ELSIF iSize<=0 THEN
    ADSLOGSTR(ADSLOG_MSGTYPE_ERROR OR ADSLOG_MSGTYPE_STRING,'CheckPointer failed due to invalid size.','');
ELSIF iGran<=0 THEN
    ADSLOGSTR(ADSLOG_MSGTYPE_ERROR OR ADSLOG_MSGTYPE_STRING,'CheckPointer failed due to invalid granularity.','');
// -> Please note that the following memory area check is time consuming:
//ELSIF F_CheckMemoryArea(pData:=ptToTest,nSize:=DINT_TO_UDINT(iSize)) = E_TcMemoryArea.Unknown THEN
//    ADSLOGSTR(ADSLOG_MSGTYPE_ERROR OR ADSLOG_MSGTYPE_STRING,'CheckPointer failed due to unknown memory area.','');
END_IF
CheckPointer := ptToTest;
{flow}

END_FUNCTION

// ---- 04_Application/Checks/CheckRangeSigned.TcPOU
// Code généré automatiquement : NE PAS MODIFIER
FUNCTION CheckRangeSigned : DINT
VAR_INPUT
	value, lower, upper: DINT;
END_VAR

// Code généré automatiquement : Il s’agit d’une proposition d’implémentation.
{noflow}
IF (value < lower) THEN
	CheckRangeSigned := lower;
ELSIF(value > upper) THEN
	CheckRangeSigned := upper;
ELSE
	CheckRangeSigned := value;
END_IF
{flow}

END_FUNCTION

// ---- 04_Application/Checks/CheckRangeUnsigned.TcPOU
// Code généré automatiquement : NE PAS MODIFIER
FUNCTION CheckRangeUnsigned : UDINT
VAR_INPUT
	value, lower, upper: UDINT;
END_VAR

// Code généré automatiquement : Il s’agit d’une proposition d’implémentation.
{noflow}
IF (value < lower) THEN
	CheckRangeUnsigned := lower;
ELSIF(value > upper) THEN
	CheckRangeUnsigned := upper;
ELSE
	CheckRangeUnsigned := value;
END_IF
{flow}

END_FUNCTION
